(* PLC project Tc2_Utilities.F_GetMaxMonthDays Demo, tc3-libraries-kb TwinCAT 3.1 *)
(* stored: creationDateTime 2026-05-11T12:00:00, modificationDateTime 2026-05-11T12:00:00 *)

PROGRAM P_Demo_F_GetMaxMonthDays
  VAR
    wYear : WORD := 2024;  (* 年份 *)
    wMonth : WORD := 2;  (* 月份 *)
    wMaxDays : WORD;  (* 该月最大天数（闰年 2 月 = 29） *)
    bRunOnce : BOOL;  (* 脉冲触发 *)
  END_VAR

// =============================================================================
// 场景：HMI 用户输入(年, 月, 日)时校验 day 不超过该月最大天数
//
// 价值：1 行调用即得月长，无需「if month in {1,3,5,7,8,10,12} ...」一长串
//
// 验证步骤：
//   1. 引用 Tc2_Utilities
//   2. 编译 + 登录 + 运行
//   3. 强制 bRunOnce := TRUE
//   4. 在线观察 wMaxDays = 29（2024 年 2 月）
//   5. wYear:=2023 重测 → wMaxDays = 28（平年 2 月）
//   6. wMonth:=0 → wMaxDays = 0（错误返回）
// =============================================================================
wMaxDays := F_GetMaxMonthDays(wYear, wMonth);
END_PROGRAM
